(* Logix 5000 project; controller PRU vendor 1 type 14 code 107 rev 20.13; software revision 20.01; part 17 of 17 *)
(* tags used below, declared in another part *)
   AFI : BOOL;
   AlarmMaster : DINT;
   ALL_SHUTDOWN_FAULTS_IOK : BOOL;
   AUTO_FWD_CMD_GON : BOOL;
   CHANGING_TOTE_1 : BOOL;
   DRYER_MODE_AUTO : BOOL;
   ENCODER_ACC : REAL;
   FEED_DWELL_DEG : INT;
   FEED_IS_DWELLING : BOOL;
   FEED_SHOT_ENABLE_Enabled : BOOL;
   FEED_SHOT_ENABLE_GON : BOOL;
   FEED_SHOT_ENABLE_GON_Tmr : TIMER;
   FEED_SHOT_ENABLE_GON_TmrONS1 : BOOL;
   FEED_SHOT_ENABLE_GON_TmrONS2 : BOOL;
   FEED_SHOT_ENABLE_ONS : BOOL;
   FEED_SHOT_ENABLE_ONSN : BOOL;
   FEED_SHOT_ENABLE_SS : BOOL;
   FEED_SHOT_ENABLE_SSN : BOOL;
   FEED_TIME : REAL;
   FEED_TIME_OFF_SEC : REAL;
   FEED_TIME_ON_SEC : REAL;
   FEED_UNWIND_THRESHOLD : INT;
   FIRST_CYCLE : BOOL;
   FWD_SCAN_COUNT : DINT;
   FWD_SCAN_COUNTING : DINT;
   FWD_SCAN_SEC : REAL;
   HMI_MIX_REV_PRESET : DINT;
   KPI : KPI;
   KPI_EnergyResetPB : BOOL;
   MIDNIGHT : BOOL;
   MIX_MODE_TIMEBASE : BOOL;
   PROCESS_SEQUENCER : INT;
   PRU_ShotEnabledTestTmr : TIMER;
   PRU_ShotEnabledTestTmrONS : BOOL;
   PRU_Status_Data : PLCStatusData;
   PYRO_CYCLE_TIME_RESET_ONS : BOOL;
   PYRO_CYCLE_TIME_RESET_SS : BOOL;
   PYRO_FWD_RUN_IOK : BOOL;
   PYRO_FWD_TON : TIMER;
   SET_PYRO_SPEED_TO_ZERO : BOOL;
   STANDBY_MODE_ION : BOOL;
   TOTAL_SCAN_COUNT : DINT;
   TOTAL_SCAN_COUNTING : DINT;
   TOTAL_SCAN_SEC : REAL;
   UTL_Status_Data : PLCStatusData;
   VFD_1_Tot : EnergyTot;   // Left Dryer
   VFD_2_Tot : EnergyTot;   // Right Dryer
   VFD_3_Tot : EnergyTot;   // Cooling Screw
   VFDS_BON : BOOL;   // DRYER VFDs HAVE BEEN COMMANDED ON FOR 1 SECOND.
   Z1L1_Tot : EnergyTot;
   Z1L2_Tot : EnergyTot;
   Z1L3_Tot : EnergyTot;
   Z2L1_Tot : EnergyTot;
   Z2L2_Tot : EnergyTot;
   Z2L3_Tot : EnergyTot;
   Z3L1_Tot : EnergyTot;
   Z3L2_Tot : EnergyTot;
   Z3L3_Tot : EnergyTot;
   Z4L1_Tot : EnergyTot;
   Z5L2_Tot : EnergyTot;
   Z6L3_Tot : EnergyTot;
   Z7L1_Tot : EnergyTot;
   Z8L2_Tot : EnergyTot;
   Z9L3_Tot : EnergyTot;
(* SCREW_CONTROL, continued *)

ROUTINE FEED_CONTROL   (* ladder *)
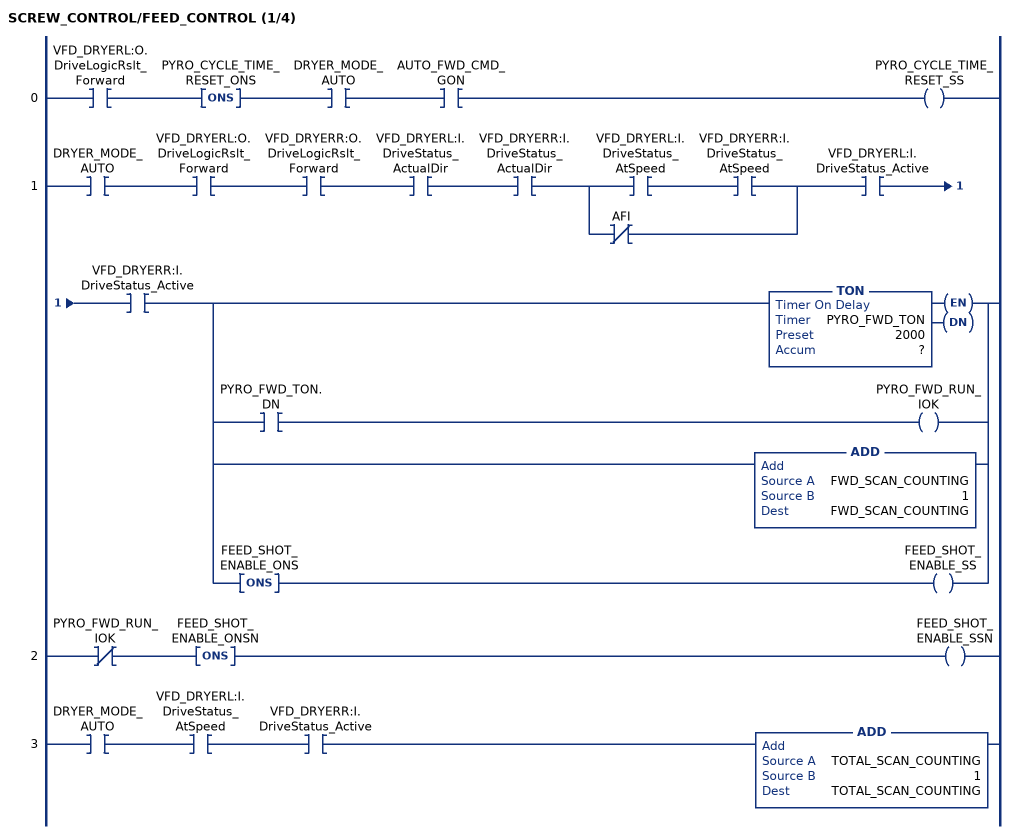
   0: XIC(VFD_DRYERL:O.DriveLogicRslt_Forward)ONS(PYRO_CYCLE_TIME_RESET_ONS)XIC(DRYER_MODE_AUTO)XIC(AUTO_FWD_CMD_GON)OTE(PYRO_CYCLE_TIME_RESET_SS);
   1: XIC(DRYER_MODE_AUTO)XIC(VFD_DRYERL:O.DriveLogicRslt_Forward)XIC(VFD_DRYERR:O.DriveLogicRslt_Forward)XIC(VFD_DRYERL:I.DriveStatus_ActualDir)XIC(VFD_DRYERR:I.DriveStatus_ActualDir)[XIC(VFD_DRYERL:I.DriveStatus_AtSpeed) XIC(VFD_DRYERR:I.DriveStatus_AtSpeed) ,XIO(AFI) ]XIC(VFD_DRYERL:I.DriveStatus_Active)XIC(VFD_DRYERR:I.DriveStatus_Active)[TON(PYRO_FWD_TON,?,?) ,XIC(PYRO_FWD_TON.DN) OTE(PYRO_FWD_RUN_IOK) ,ADD(FWD_SCAN_COUNTING,1,FWD_SCAN_COUNTING) ,ONS(FEED_SHOT_ENABLE_ONS) OTE(FEED_SHOT_ENABLE_SS) ];
   2: XIO(PYRO_FWD_RUN_IOK)ONS(FEED_SHOT_ENABLE_ONSN)OTE(FEED_SHOT_ENABLE_SSN);
   3: XIC(DRYER_MODE_AUTO)XIC(VFD_DRYERL:I.DriveStatus_AtSpeed)XIC(VFD_DRYERR:I.DriveStatus_Active)ADD(TOTAL_SCAN_COUNTING,1,TOTAL_SCAN_COUNTING);
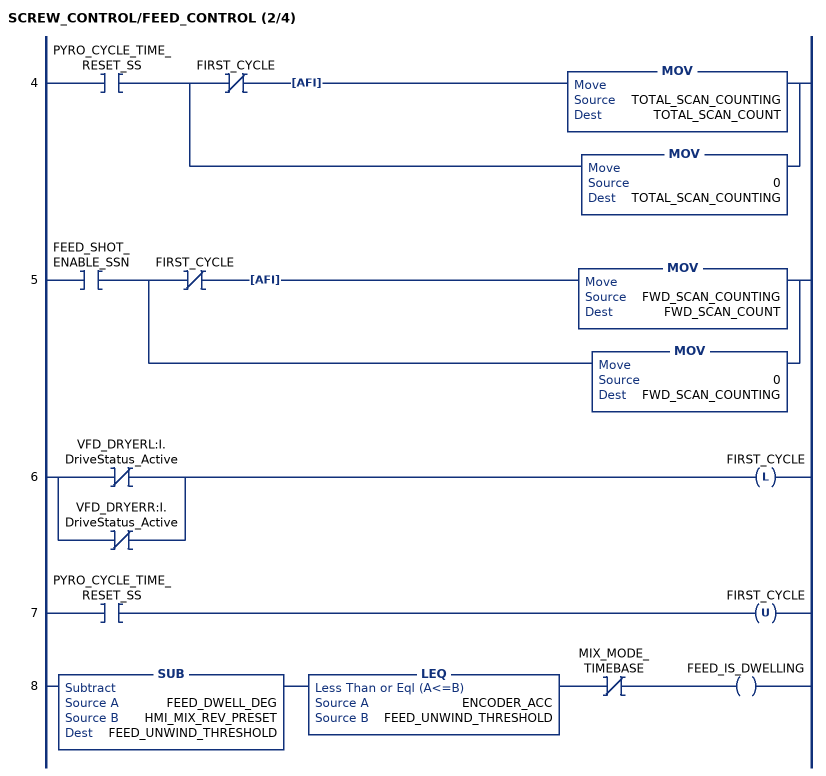
   4: XIC(PYRO_CYCLE_TIME_RESET_SS)[XIO(FIRST_CYCLE) AFI() MOV(TOTAL_SCAN_COUNTING,TOTAL_SCAN_COUNT) ,MOV(0,TOTAL_SCAN_COUNTING) ];
   5: XIC(FEED_SHOT_ENABLE_SSN)[XIO(FIRST_CYCLE) AFI() MOV(FWD_SCAN_COUNTING,FWD_SCAN_COUNT) ,MOV(0,FWD_SCAN_COUNTING) ];
   6: [XIO(VFD_DRYERL:I.DriveStatus_Active) ,XIO(VFD_DRYERR:I.DriveStatus_Active) ]OTL(FIRST_CYCLE);
   7: XIC(PYRO_CYCLE_TIME_RESET_SS)OTU(FIRST_CYCLE);
   8: SUB(FEED_DWELL_DEG,HMI_MIX_REV_PRESET,FEED_UNWIND_THRESHOLD)LEQ(ENCODER_ACC,FEED_UNWIND_THRESHOLD)XIO(MIX_MODE_TIMEBASE)OTE(FEED_IS_DWELLING);
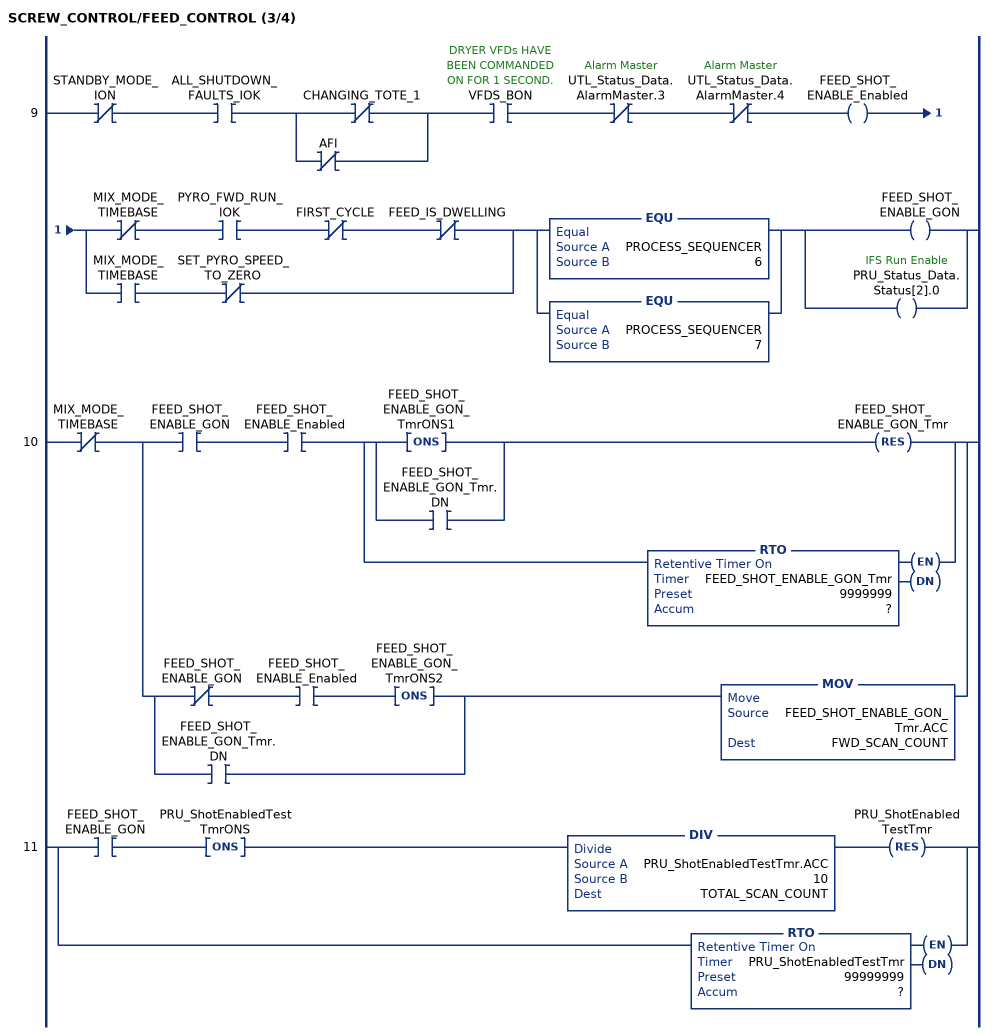
   9: XIO(STANDBY_MODE_ION)XIC(ALL_SHUTDOWN_FAULTS_IOK)[XIO(CHANGING_TOTE_1) ,XIO(AFI) ]XIC(VFDS_BON)XIO(UTL_Status_Data.AlarmMaster.3)XIO(UTL_Status_Data.AlarmMaster.4)OTE(FEED_SHOT_ENABLE_Enabled)[XIO(MIX_MODE_TIMEBASE) XIC(PYRO_FWD_RUN_IOK) XIO(FIRST_CYCLE) XIO(FEED_IS_DWELLING) ,XIC(MIX_MODE_TIMEBASE) XIO(SET_PYRO_SPEED_TO_ZERO) ][EQU(PROCESS_SEQUENCER,6) ,EQU(PROCESS_SEQUENCER,7) ][OTE(FEED_SHOT_ENABLE_GON) ,OTE(PRU_Status_Data.Status[2].0) ];
   10: XIO(MIX_MODE_TIMEBASE)[XIC(FEED_SHOT_ENABLE_GON) XIC(FEED_SHOT_ENABLE_Enabled) [[ONS(FEED_SHOT_ENABLE_GON_TmrONS1) ,XIC(FEED_SHOT_ENABLE_GON_Tmr.DN) ] RES(FEED_SHOT_ENABLE_GON_Tmr) ,RTO(FEED_SHOT_ENABLE_GON_Tmr,?,?) ] ,[XIO(FEED_SHOT_ENABLE_GON) XIC(FEED_SHOT_ENABLE_Enabled) ONS(FEED_SHOT_ENABLE_GON_TmrONS2) ,XIC(FEED_SHOT_ENABLE_GON_Tmr.DN) ] MOV(FEED_SHOT_ENABLE_GON_Tmr.ACC,FWD_SCAN_COUNT) ];
   11: [XIC(FEED_SHOT_ENABLE_GON) ONS(PRU_ShotEnabledTestTmrONS) DIV(PRU_ShotEnabledTestTmr.ACC,10,TOTAL_SCAN_COUNT) RES(PRU_ShotEnabledTestTmr) ,RTO(PRU_ShotEnabledTestTmr,?,?) ];
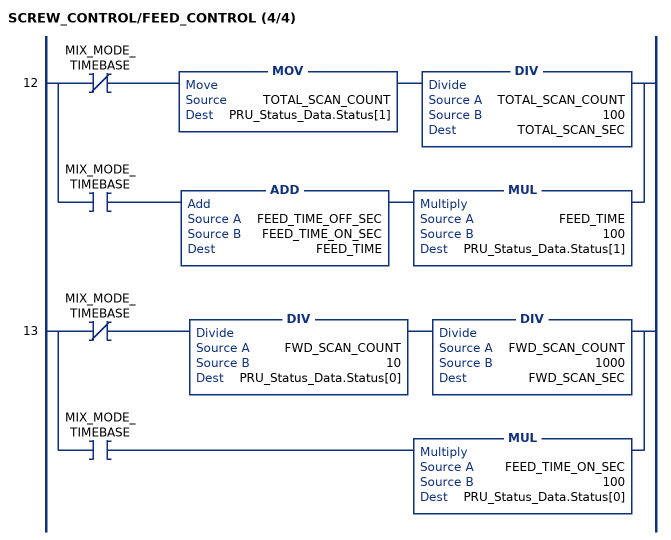
   12: [XIO(MIX_MODE_TIMEBASE) MOV(TOTAL_SCAN_COUNT,PRU_Status_Data.Status[1]) DIV(TOTAL_SCAN_COUNT,100,TOTAL_SCAN_SEC) ,XIC(MIX_MODE_TIMEBASE) ADD(FEED_TIME_OFF_SEC,FEED_TIME_ON_SEC,FEED_TIME) MUL(FEED_TIME,100,PRU_Status_Data.Status[1]) ];
   13: [XIO(MIX_MODE_TIMEBASE) DIV(FWD_SCAN_COUNT,10,PRU_Status_Data.Status[0]) DIV(FWD_SCAN_COUNT,1000,FWD_SCAN_SEC) ,XIC(MIX_MODE_TIMEBASE) MUL(FEED_TIME_ON_SEC,100,PRU_Status_Data.Status[0]) ];
END_ROUTINE
END_PROGRAM

PROGRAM Totalizers   (* main routine MainRoutine *)
VAR
   AITot_VFD1 : AI_Totalizer := (Input := 5.23152, SampleTimerSP := 1, TimeBase := 3, MinimumInc := 1.0, IDP := 2, RollOver := 999999999, NonResetTotal := 618304, TodayTotal := 1933, YestTotal := 4297, ResetTotal := 497307);
   AITot_VFD2 : AI_Totalizer := (Input := 5.3976, SampleTimerSP := 1, TimeBase := 3, MinimumInc := 1.0, IDP := 2, RollOver := 999999999, NonResetTotal := 632266, TodayTotal := 1996, YestTotal := 4422, ResetTotal := 509519);
   AITot_VFD3 : AI_Totalizer := (Input := 1.5943679, SampleTimerSP := 1, TimeBase := 3, MinimumInc := 1.0, IDP := 2, RollOver := 999999999, NonResetTotal := 173015, TodayTotal := 587, YestTotal := 1277, ResetTotal := 140164);
   AITot_Z1L1 : AI_Totalizer := (Input := 1.689711, SampleTimerSP := 1, TimeBase := 3, MinimumInc := 1.0, IDP := 2, RollOver := 999999999, NonResetTotal := 472353, TodayTotal := 130, YestTotal := 3764, ResetTotal := 404849);
   AITot_Z1L2 : AI_Totalizer := (Input := 0.03052023, SampleTimerSP := 1, TimeBase := 3, MinimumInc := 1.0, IDP := 2, RollOver := 999999999, NonResetTotal := 457837, TodayTotal := 130, YestTotal := 3741, ResetTotal := 457837);
   AITot_Z1L3 : AI_Totalizer := (Input := 0.03052023, SampleTimerSP := 1, TimeBase := 3, MinimumInc := 1.0, IDP := 2, RollOver := 999999999, NonResetTotal := 456822, TodayTotal := 160, YestTotal := 4321, ResetTotal := 390415);
   AITot_Z2L1 : AI_Totalizer := (Input := 1.2069364, SampleTimerSP := 1, TimeBase := 3, MinimumInc := 1.0, IDP := 2, RollOver := 999999999, NonResetTotal := 262631, TodayTotal := 198, YestTotal := 2727, ResetTotal := 202203);
   AITot_Z2L2 : AI_Totalizer := (Input := 0.033294797, SampleTimerSP := 1, TimeBase := 3, MinimumInc := 1.0, IDP := 2, RollOver := 999999999, NonResetTotal := 260774, TodayTotal := 195, YestTotal := 2658, ResetTotal := 201494);
   AITot_Z2L3 : AI_Totalizer := (Input := 1.2873988, SampleTimerSP := 1, TimeBase := 3, MinimumInc := 1.0, IDP := 2, RollOver := 999999999, NonResetTotal := 261254, TodayTotal := 195, YestTotal := 2685, ResetTotal := 201639);
   AITot_Z3L1 : AI_Totalizer := (Input := 0.8323699, SampleTimerSP := 1, TimeBase := 3, MinimumInc := 1.0, IDP := 2, RollOver := 999999999, NonResetTotal := 191746, TodayTotal := 428, YestTotal := 2124, ResetTotal := 154486);
   AITot_Z3L2 : AI_Totalizer := (Input := 0.88508666, SampleTimerSP := 1, TimeBase := 3, MinimumInc := 1.0, IDP := 2, RollOver := 999999999, NonResetTotal := 197557, TodayTotal := 352, YestTotal := 1665, ResetTotal := 160053);
   AITot_Z3L3 : AI_Totalizer := (Input := 0.59930634, SampleTimerSP := 1, TimeBase := 3, MinimumInc := 1.0, IDP := 2, RollOver := 999999999, NonResetTotal := 197140, TodayTotal := 341, YestTotal := 1652, ResetTotal := 160368);
   AITot_Z4L1 : AI_Totalizer := (Input := 0.88508666, SampleTimerSP := 1, TimeBase := 3, MinimumInc := 1.0, IDP := 2, RollOver := 999999999, NonResetTotal := 314322, TodayTotal := 64, YestTotal := 1698, ResetTotal := 297528);
   AITot_Z5L2 : AI_Totalizer := (Input := 0.03052023, SampleTimerSP := 1, TimeBase := 3, MinimumInc := 1.0, IDP := 2, RollOver := 999999999, NonResetTotal := 574405, TodayTotal := 368, YestTotal := 5145, ResetTotal := 490444);
   AITot_Z6L3 : AI_Totalizer := (Input := 0.30797687, SampleTimerSP := 1, TimeBase := 3, MinimumInc := 1.0, IDP := 2, RollOver := 999999999, NonResetTotal := 104261, TodayTotal := 197, YestTotal := 2603, ResetTotal := 99809);
   AITot_Z7L1 : AI_Totalizer := (Input := 0.03052023, SampleTimerSP := 1, TimeBase := 3, MinimumInc := 1.0, IDP := 2, RollOver := 999999999, NonResetTotal := 390081, TodayTotal := 454, YestTotal := 4326, ResetTotal := 301917);
   AITot_Z8L2 : AI_Totalizer := (Input := 5.041387, SampleTimerSP := 1, TimeBase := 3, MinimumInc := 1.0, IDP := 2, RollOver := 999999999, NonResetTotal := 336435, TodayTotal := 1724, YestTotal := 5854, ResetTotal := 321398);
   AITot_Z9L3 : AI_Totalizer := (Input := 5.6684394, SampleTimerSP := 1, TimeBase := 3, MinimumInc := 1.0, IDP := 2, RollOver := 999999999, NonResetTotal := 446178, TodayTotal := 1624, YestTotal := 4125, ResetTotal := 368110);
   ResetTotalizersONS : BOOL;
END_VAR

ROUTINE MainRoutine   (* ladder *)
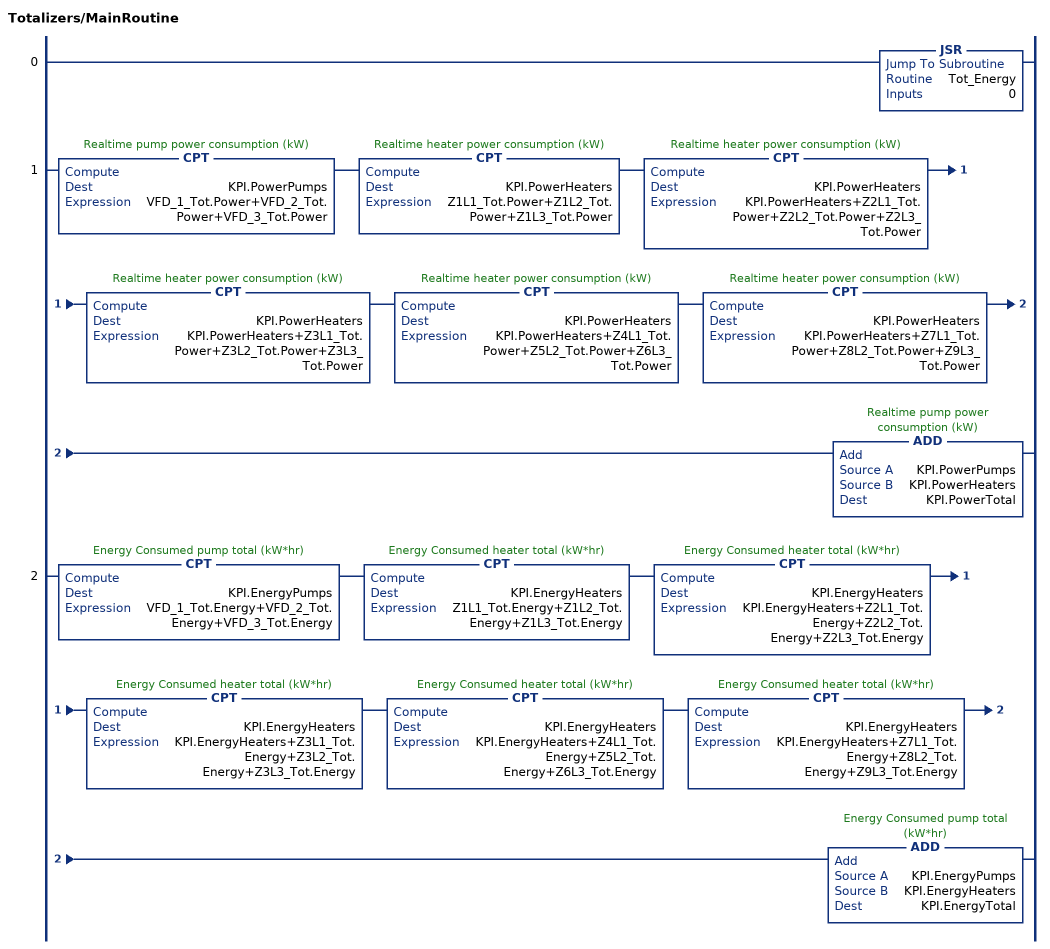
   0: JSR(Tot_Energy,0);
   1: CPT(KPI.PowerPumps,VFD_1_Tot.Power+VFD_2_Tot.Power+VFD_3_Tot.Power)CPT(KPI.PowerHeaters,Z1L1_Tot.Power+Z1L2_Tot.Power+Z1L3_Tot.Power)CPT(KPI.PowerHeaters,KPI.PowerHeaters+Z2L1_Tot.Power+Z2L2_Tot.Power+Z2L3_Tot.Power)CPT(KPI.PowerHeaters,KPI.PowerHeaters+Z3L1_Tot.Power+Z3L2_Tot.Power+Z3L3_Tot.Power)CPT(KPI.PowerHeaters,KPI.PowerHeaters+Z4L1_Tot.Power+Z5L2_Tot.Power+Z6L3_Tot.Power)CPT(KPI.PowerHeaters,KPI.PowerHeaters+Z7L1_Tot.Power+Z8L2_Tot.Power+Z9L3_Tot.Power)ADD(KPI.PowerPumps,KPI.PowerHeaters,KPI.PowerTotal);
   2: CPT(KPI.EnergyPumps,VFD_1_Tot.Energy+VFD_2_Tot.Energy+VFD_3_Tot.Energy)CPT(KPI.EnergyHeaters,Z1L1_Tot.Energy+Z1L2_Tot.Energy+Z1L3_Tot.Energy)CPT(KPI.EnergyHeaters,KPI.EnergyHeaters+Z2L1_Tot.Energy+Z2L2_Tot.Energy+Z2L3_Tot.Energy)CPT(KPI.EnergyHeaters,KPI.EnergyHeaters+Z3L1_Tot.Energy+Z3L2_Tot.Energy+Z3L3_Tot.Energy)CPT(KPI.EnergyHeaters,KPI.EnergyHeaters+Z4L1_Tot.Energy+Z5L2_Tot.Energy+Z6L3_Tot.Energy)CPT(KPI.EnergyHeaters,KPI.EnergyHeaters+Z7L1_Tot.Energy+Z8L2_Tot.Energy+Z9L3_Tot.Energy)ADD(KPI.EnergyPumps,KPI.EnergyHeaters,KPI.EnergyTotal);
END_ROUTINE

ROUTINE Tot_Energy   (* ladder *)
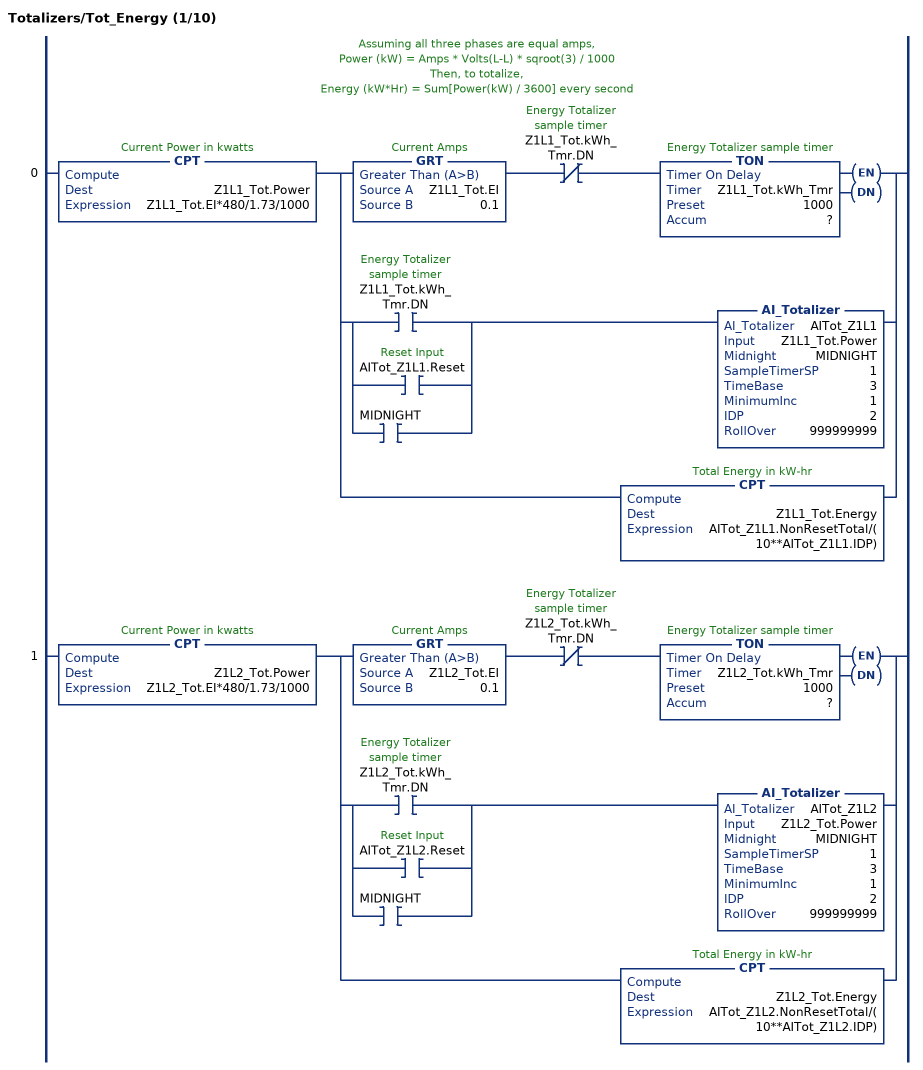
   // Assuming all three phases are equal amps,
   // Power (kW) = Amps * Volts(L-L) * sqroot(3) / 1000
   // Then, to totalize,
   // Energy (kW*Hr) = Sum[Power(kW) / 3600] every second
   0: CPT(Z1L1_Tot.Power,Z1L1_Tot.EI*480/1.73/1000)[GRT(Z1L1_Tot.EI,0.1) XIO(Z1L1_Tot.kWh_Tmr.DN) TON(Z1L1_Tot.kWh_Tmr,?,?) ,[XIC(Z1L1_Tot.kWh_Tmr.DN) ,XIC(AITot_Z1L1.Reset) ,XIC(MIDNIGHT) ] AI_Totalizer(AITot_Z1L1,Z1L1_Tot.Power,MIDNIGHT,1,3,1,2,999999999) ,CPT(Z1L1_Tot.Energy,AITot_Z1L1.NonResetTotal/(10**AITot_Z1L1.IDP)) ];
   1: CPT(Z1L2_Tot.Power,Z1L2_Tot.EI*480/1.73/1000)[GRT(Z1L2_Tot.EI,0.1) XIO(Z1L2_Tot.kWh_Tmr.DN) TON(Z1L2_Tot.kWh_Tmr,?,?) ,[XIC(Z1L2_Tot.kWh_Tmr.DN) ,XIC(AITot_Z1L2.Reset) ,XIC(MIDNIGHT) ] AI_Totalizer(AITot_Z1L2,Z1L2_Tot.Power,MIDNIGHT,1,3,1,2,999999999) ,CPT(Z1L2_Tot.Energy,AITot_Z1L2.NonResetTotal/(10**AITot_Z1L2.IDP)) ];
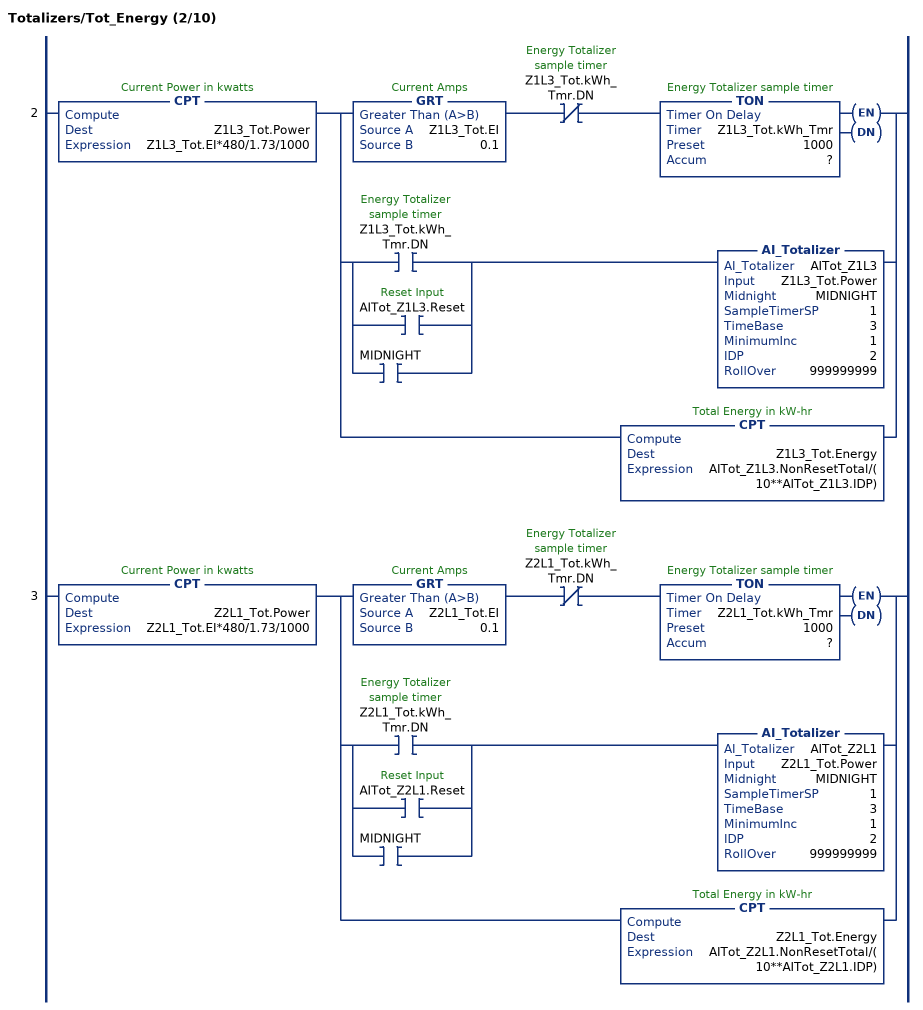
   2: CPT(Z1L3_Tot.Power,Z1L3_Tot.EI*480/1.73/1000)[GRT(Z1L3_Tot.EI,0.1) XIO(Z1L3_Tot.kWh_Tmr.DN) TON(Z1L3_Tot.kWh_Tmr,?,?) ,[XIC(Z1L3_Tot.kWh_Tmr.DN) ,XIC(AITot_Z1L3.Reset) ,XIC(MIDNIGHT) ] AI_Totalizer(AITot_Z1L3,Z1L3_Tot.Power,MIDNIGHT,1,3,1,2,999999999) ,CPT(Z1L3_Tot.Energy,AITot_Z1L3.NonResetTotal/(10**AITot_Z1L3.IDP)) ];
   3: CPT(Z2L1_Tot.Power,Z2L1_Tot.EI*480/1.73/1000)[GRT(Z2L1_Tot.EI,0.1) XIO(Z2L1_Tot.kWh_Tmr.DN) TON(Z2L1_Tot.kWh_Tmr,?,?) ,[XIC(Z2L1_Tot.kWh_Tmr.DN) ,XIC(AITot_Z2L1.Reset) ,XIC(MIDNIGHT) ] AI_Totalizer(AITot_Z2L1,Z2L1_Tot.Power,MIDNIGHT,1,3,1,2,999999999) ,CPT(Z2L1_Tot.Energy,AITot_Z2L1.NonResetTotal/(10**AITot_Z2L1.IDP)) ];
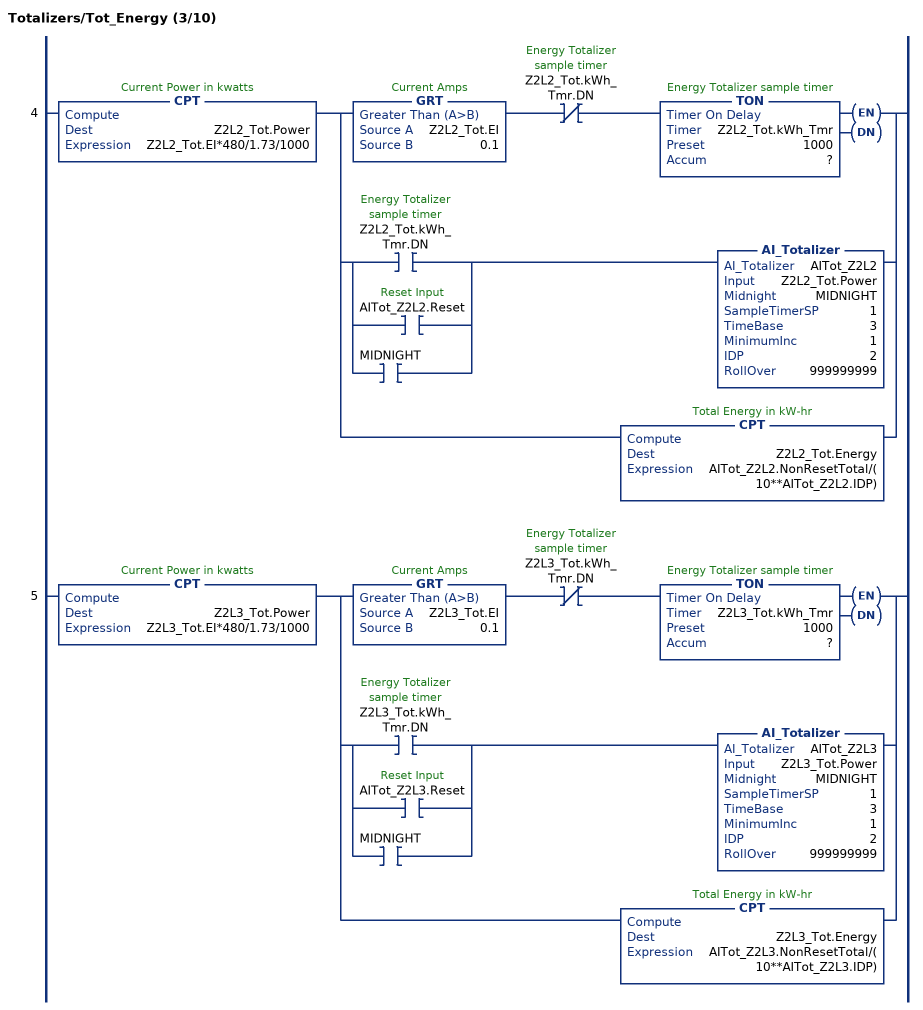
   4: CPT(Z2L2_Tot.Power,Z2L2_Tot.EI*480/1.73/1000)[GRT(Z2L2_Tot.EI,0.1) XIO(Z2L2_Tot.kWh_Tmr.DN) TON(Z2L2_Tot.kWh_Tmr,?,?) ,[XIC(Z2L2_Tot.kWh_Tmr.DN) ,XIC(AITot_Z2L2.Reset) ,XIC(MIDNIGHT) ] AI_Totalizer(AITot_Z2L2,Z2L2_Tot.Power,MIDNIGHT,1,3,1,2,999999999) ,CPT(Z2L2_Tot.Energy,AITot_Z2L2.NonResetTotal/(10**AITot_Z2L2.IDP)) ];
   5: CPT(Z2L3_Tot.Power,Z2L3_Tot.EI*480/1.73/1000)[GRT(Z2L3_Tot.EI,0.1) XIO(Z2L3_Tot.kWh_Tmr.DN) TON(Z2L3_Tot.kWh_Tmr,?,?) ,[XIC(Z2L3_Tot.kWh_Tmr.DN) ,XIC(AITot_Z2L3.Reset) ,XIC(MIDNIGHT) ] AI_Totalizer(AITot_Z2L3,Z2L3_Tot.Power,MIDNIGHT,1,3,1,2,999999999) ,CPT(Z2L3_Tot.Energy,AITot_Z2L3.NonResetTotal/(10**AITot_Z2L3.IDP)) ];
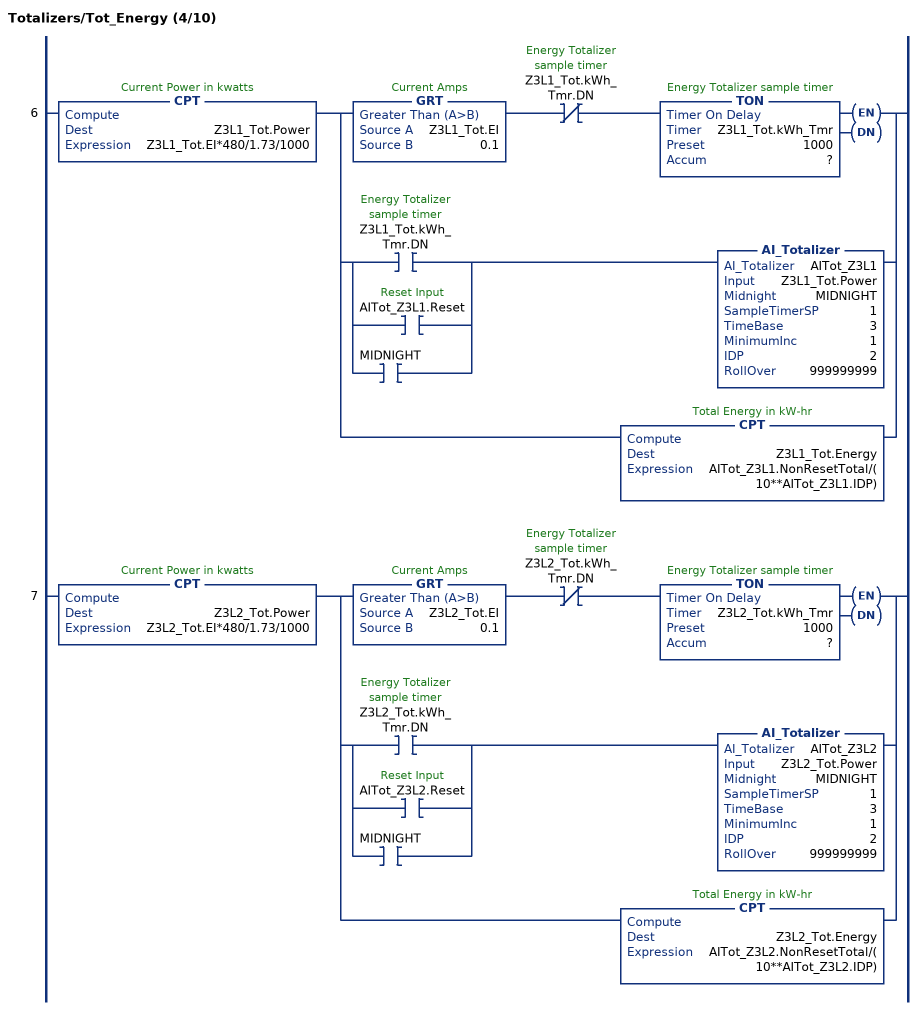
   6: CPT(Z3L1_Tot.Power,Z3L1_Tot.EI*480/1.73/1000)[GRT(Z3L1_Tot.EI,0.1) XIO(Z3L1_Tot.kWh_Tmr.DN) TON(Z3L1_Tot.kWh_Tmr,?,?) ,[XIC(Z3L1_Tot.kWh_Tmr.DN) ,XIC(AITot_Z3L1.Reset) ,XIC(MIDNIGHT) ] AI_Totalizer(AITot_Z3L1,Z3L1_Tot.Power,MIDNIGHT,1,3,1,2,999999999) ,CPT(Z3L1_Tot.Energy,AITot_Z3L1.NonResetTotal/(10**AITot_Z3L1.IDP)) ];
   7: CPT(Z3L2_Tot.Power,Z3L2_Tot.EI*480/1.73/1000)[GRT(Z3L2_Tot.EI,0.1) XIO(Z3L2_Tot.kWh_Tmr.DN) TON(Z3L2_Tot.kWh_Tmr,?,?) ,[XIC(Z3L2_Tot.kWh_Tmr.DN) ,XIC(AITot_Z3L2.Reset) ,XIC(MIDNIGHT) ] AI_Totalizer(AITot_Z3L2,Z3L2_Tot.Power,MIDNIGHT,1,3,1,2,999999999) ,CPT(Z3L2_Tot.Energy,AITot_Z3L2.NonResetTotal/(10**AITot_Z3L2.IDP)) ];
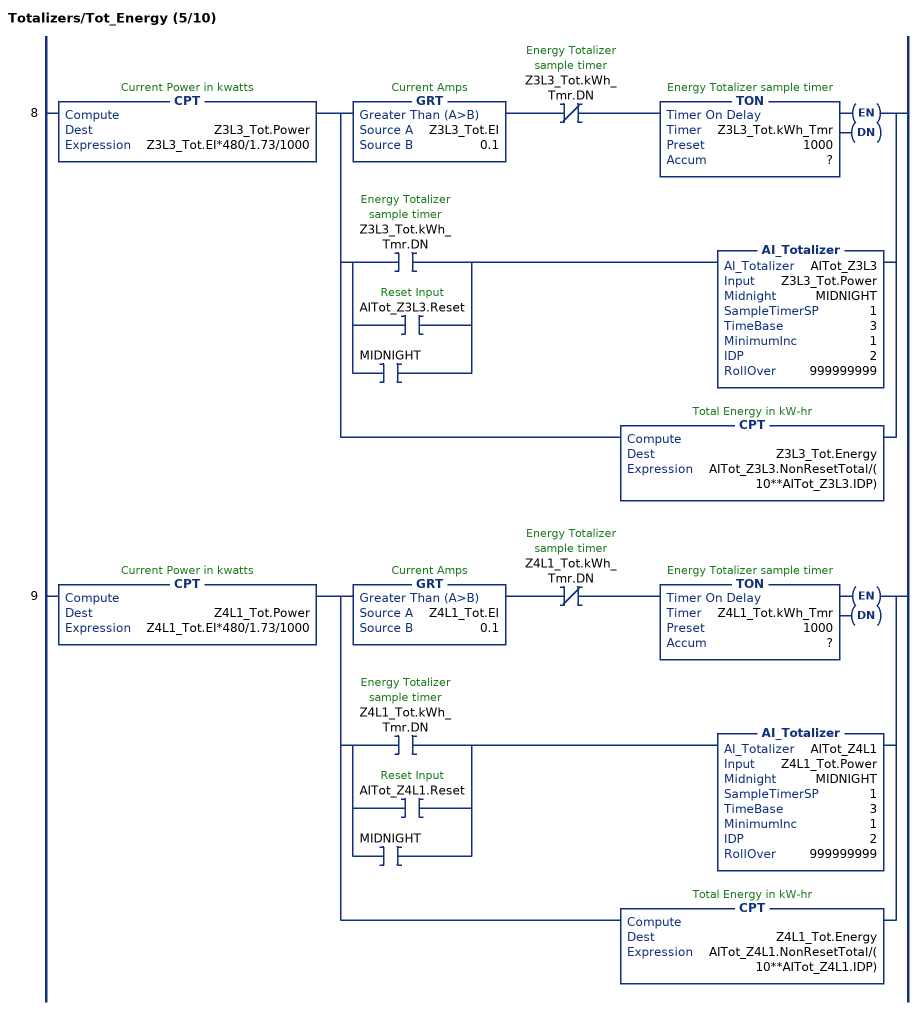
   8: CPT(Z3L3_Tot.Power,Z3L3_Tot.EI*480/1.73/1000)[GRT(Z3L3_Tot.EI,0.1) XIO(Z3L3_Tot.kWh_Tmr.DN) TON(Z3L3_Tot.kWh_Tmr,?,?) ,[XIC(Z3L3_Tot.kWh_Tmr.DN) ,XIC(AITot_Z3L3.Reset) ,XIC(MIDNIGHT) ] AI_Totalizer(AITot_Z3L3,Z3L3_Tot.Power,MIDNIGHT,1,3,1,2,999999999) ,CPT(Z3L3_Tot.Energy,AITot_Z3L3.NonResetTotal/(10**AITot_Z3L3.IDP)) ];
   9: CPT(Z4L1_Tot.Power,Z4L1_Tot.EI*480/1.73/1000)[GRT(Z4L1_Tot.EI,0.1) XIO(Z4L1_Tot.kWh_Tmr.DN) TON(Z4L1_Tot.kWh_Tmr,?,?) ,[XIC(Z4L1_Tot.kWh_Tmr.DN) ,XIC(AITot_Z4L1.Reset) ,XIC(MIDNIGHT) ] AI_Totalizer(AITot_Z4L1,Z4L1_Tot.Power,MIDNIGHT,1,3,1,2,999999999) ,CPT(Z4L1_Tot.Energy,AITot_Z4L1.NonResetTotal/(10**AITot_Z4L1.IDP)) ];
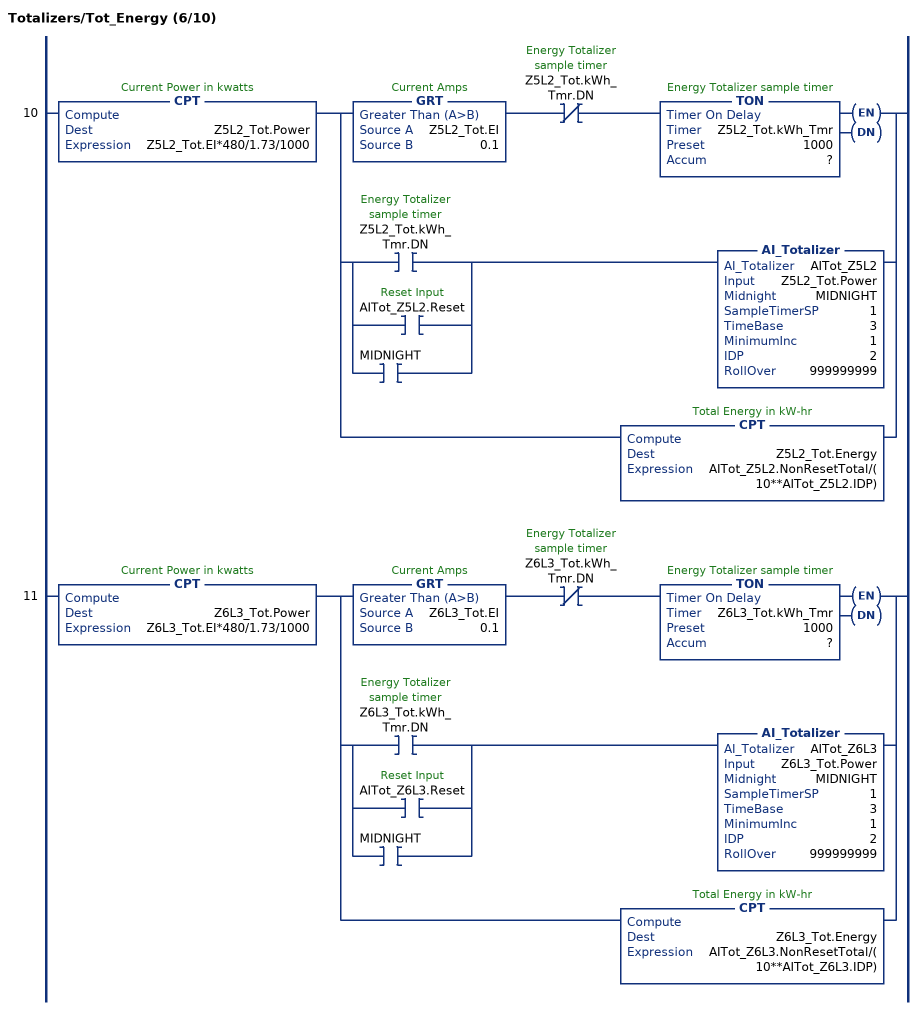
   10: CPT(Z5L2_Tot.Power,Z5L2_Tot.EI*480/1.73/1000)[GRT(Z5L2_Tot.EI,0.1) XIO(Z5L2_Tot.kWh_Tmr.DN) TON(Z5L2_Tot.kWh_Tmr,?,?) ,[XIC(Z5L2_Tot.kWh_Tmr.DN) ,XIC(AITot_Z5L2.Reset) ,XIC(MIDNIGHT) ] AI_Totalizer(AITot_Z5L2,Z5L2_Tot.Power,MIDNIGHT,1,3,1,2,999999999) ,CPT(Z5L2_Tot.Energy,AITot_Z5L2.NonResetTotal/(10**AITot_Z5L2.IDP)) ];
   11: CPT(Z6L3_Tot.Power,Z6L3_Tot.EI*480/1.73/1000)[GRT(Z6L3_Tot.EI,0.1) XIO(Z6L3_Tot.kWh_Tmr.DN) TON(Z6L3_Tot.kWh_Tmr,?,?) ,[XIC(Z6L3_Tot.kWh_Tmr.DN) ,XIC(AITot_Z6L3.Reset) ,XIC(MIDNIGHT) ] AI_Totalizer(AITot_Z6L3,Z6L3_Tot.Power,MIDNIGHT,1,3,1,2,999999999) ,CPT(Z6L3_Tot.Energy,AITot_Z6L3.NonResetTotal/(10**AITot_Z6L3.IDP)) ];
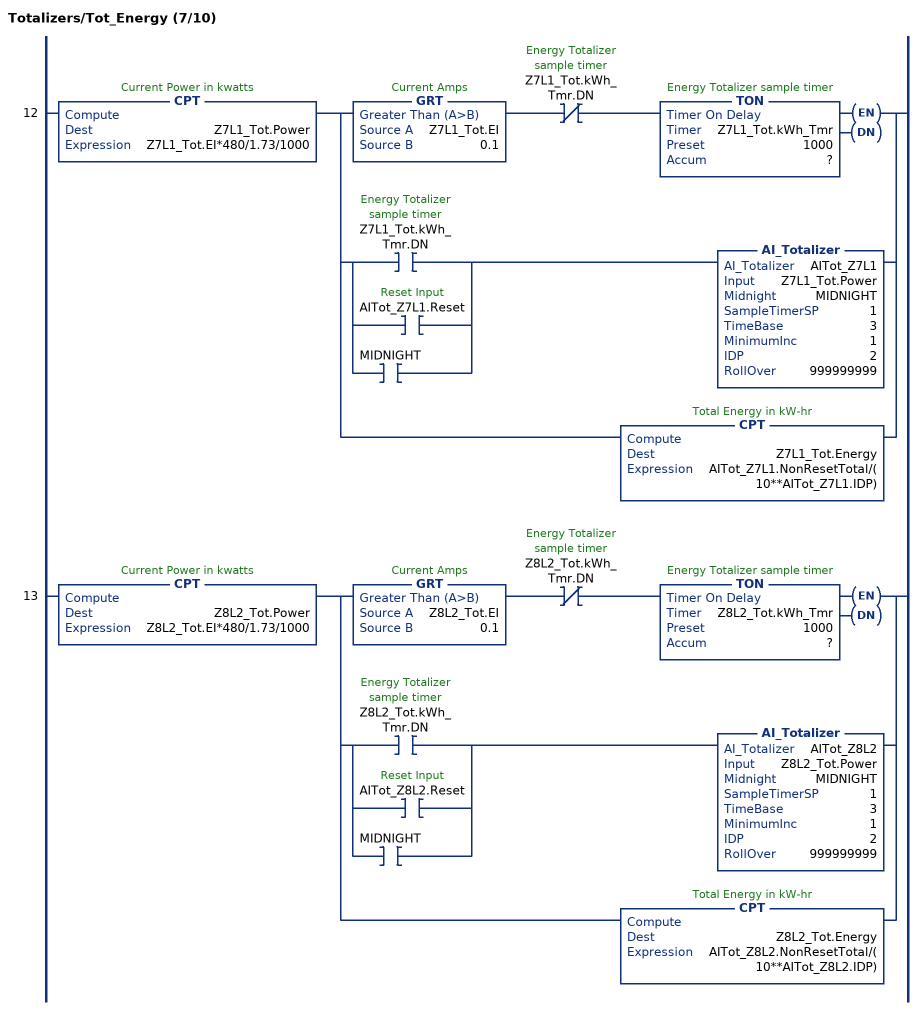
   12: CPT(Z7L1_Tot.Power,Z7L1_Tot.EI*480/1.73/1000)[GRT(Z7L1_Tot.EI,0.1) XIO(Z7L1_Tot.kWh_Tmr.DN) TON(Z7L1_Tot.kWh_Tmr,?,?) ,[XIC(Z7L1_Tot.kWh_Tmr.DN) ,XIC(AITot_Z7L1.Reset) ,XIC(MIDNIGHT) ] AI_Totalizer(AITot_Z7L1,Z7L1_Tot.Power,MIDNIGHT,1,3,1,2,999999999) ,CPT(Z7L1_Tot.Energy,AITot_Z7L1.NonResetTotal/(10**AITot_Z7L1.IDP)) ];
   13: CPT(Z8L2_Tot.Power,Z8L2_Tot.EI*480/1.73/1000)[GRT(Z8L2_Tot.EI,0.1) XIO(Z8L2_Tot.kWh_Tmr.DN) TON(Z8L2_Tot.kWh_Tmr,?,?) ,[XIC(Z8L2_Tot.kWh_Tmr.DN) ,XIC(AITot_Z8L2.Reset) ,XIC(MIDNIGHT) ] AI_Totalizer(AITot_Z8L2,Z8L2_Tot.Power,MIDNIGHT,1,3,1,2,999999999) ,CPT(Z8L2_Tot.Energy,AITot_Z8L2.NonResetTotal/(10**AITot_Z8L2.IDP)) ];
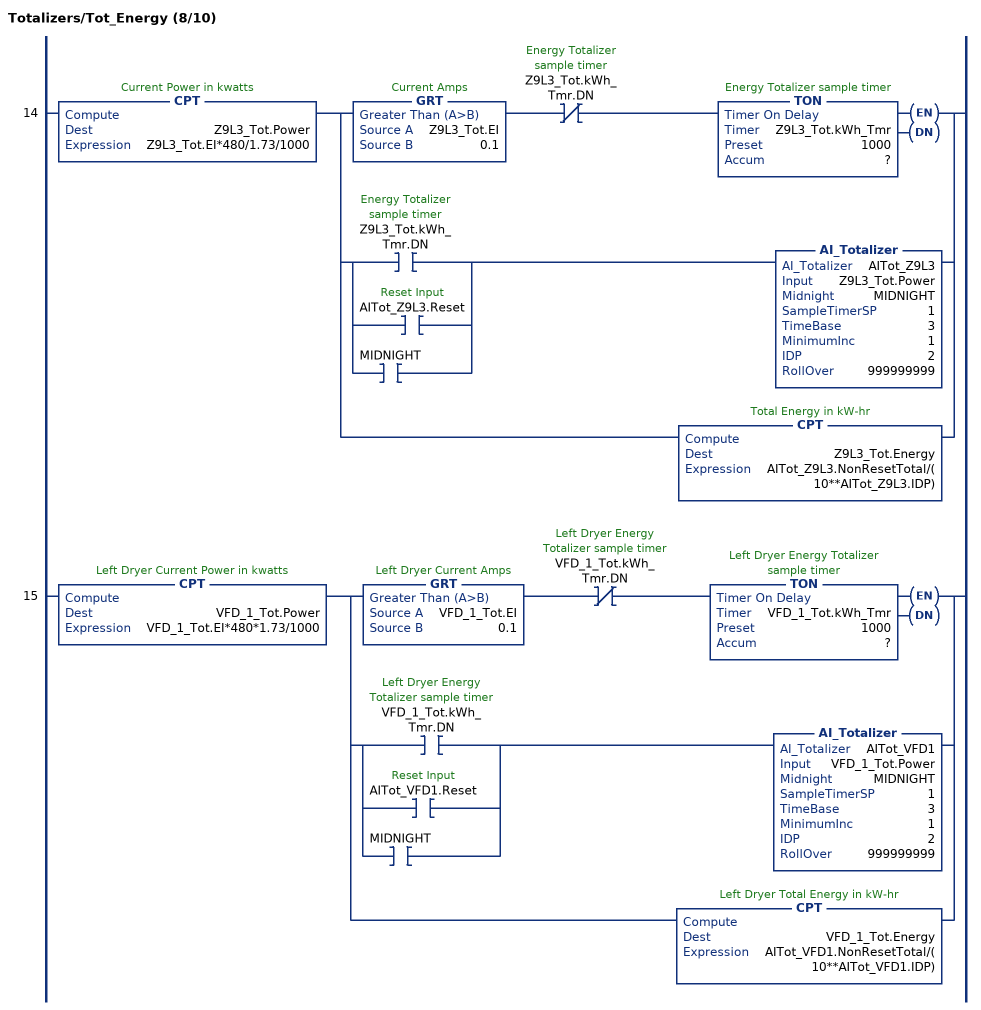
   14: CPT(Z9L3_Tot.Power,Z9L3_Tot.EI*480/1.73/1000)[GRT(Z9L3_Tot.EI,0.1) XIO(Z9L3_Tot.kWh_Tmr.DN) TON(Z9L3_Tot.kWh_Tmr,?,?) ,[XIC(Z9L3_Tot.kWh_Tmr.DN) ,XIC(AITot_Z9L3.Reset) ,XIC(MIDNIGHT) ] AI_Totalizer(AITot_Z9L3,Z9L3_Tot.Power,MIDNIGHT,1,3,1,2,999999999) ,CPT(Z9L3_Tot.Energy,AITot_Z9L3.NonResetTotal/(10**AITot_Z9L3.IDP)) ];
   15: CPT(VFD_1_Tot.Power,VFD_1_Tot.EI*480*1.73/1000)[GRT(VFD_1_Tot.EI,0.1) XIO(VFD_1_Tot.kWh_Tmr.DN) TON(VFD_1_Tot.kWh_Tmr,?,?) ,[XIC(VFD_1_Tot.kWh_Tmr.DN) ,XIC(AITot_VFD1.Reset) ,XIC(MIDNIGHT) ] AI_Totalizer(AITot_VFD1,VFD_1_Tot.Power,MIDNIGHT,1,3,1,2,999999999) ,CPT(VFD_1_Tot.Energy,AITot_VFD1.NonResetTotal/(10**AITot_VFD1.IDP)) ];
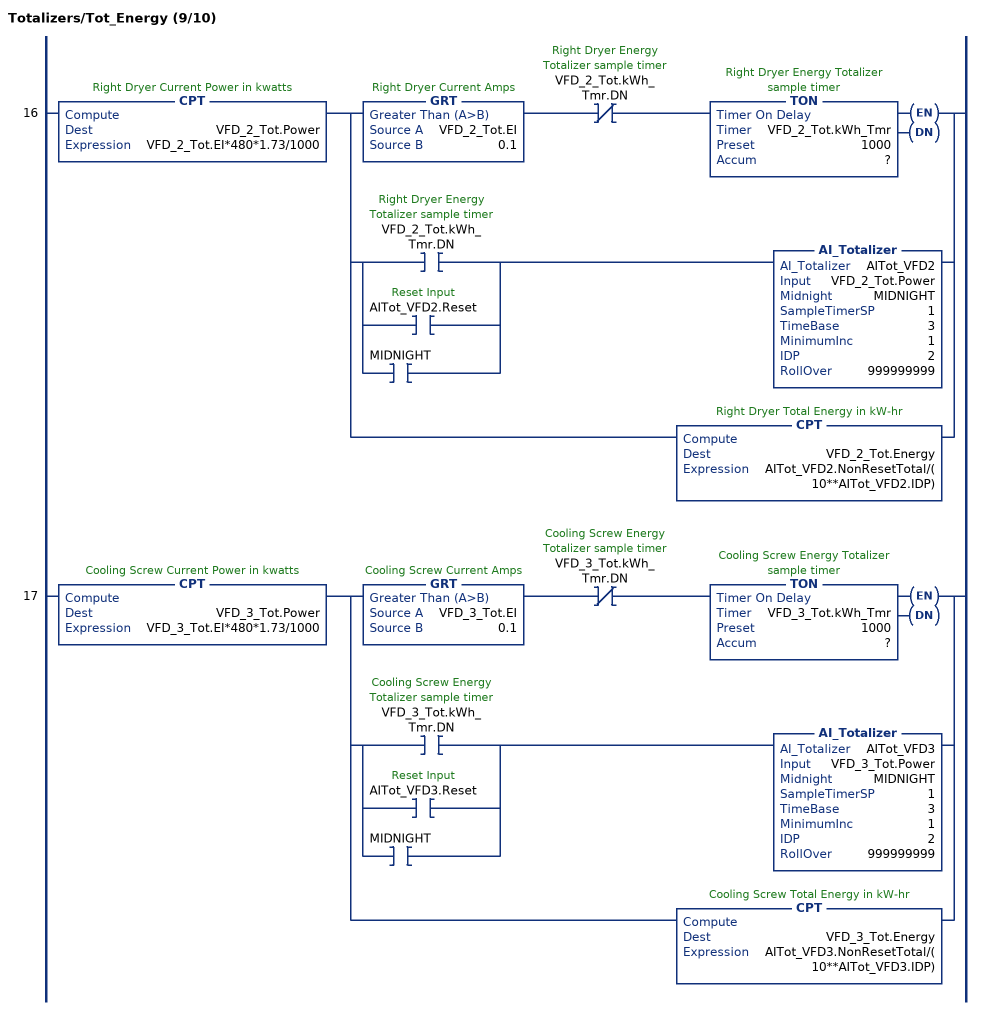
   16: CPT(VFD_2_Tot.Power,VFD_2_Tot.EI*480*1.73/1000)[GRT(VFD_2_Tot.EI,0.1) XIO(VFD_2_Tot.kWh_Tmr.DN) TON(VFD_2_Tot.kWh_Tmr,?,?) ,[XIC(VFD_2_Tot.kWh_Tmr.DN) ,XIC(AITot_VFD2.Reset) ,XIC(MIDNIGHT) ] AI_Totalizer(AITot_VFD2,VFD_2_Tot.Power,MIDNIGHT,1,3,1,2,999999999) ,CPT(VFD_2_Tot.Energy,AITot_VFD2.NonResetTotal/(10**AITot_VFD2.IDP)) ];
   17: CPT(VFD_3_Tot.Power,VFD_3_Tot.EI*480*1.73/1000)[GRT(VFD_3_Tot.EI,0.1) XIO(VFD_3_Tot.kWh_Tmr.DN) TON(VFD_3_Tot.kWh_Tmr,?,?) ,[XIC(VFD_3_Tot.kWh_Tmr.DN) ,XIC(AITot_VFD3.Reset) ,XIC(MIDNIGHT) ] AI_Totalizer(AITot_VFD3,VFD_3_Tot.Power,MIDNIGHT,1,3,1,2,999999999) ,CPT(VFD_3_Tot.Energy,AITot_VFD3.NonResetTotal/(10**AITot_VFD3.IDP)) ];
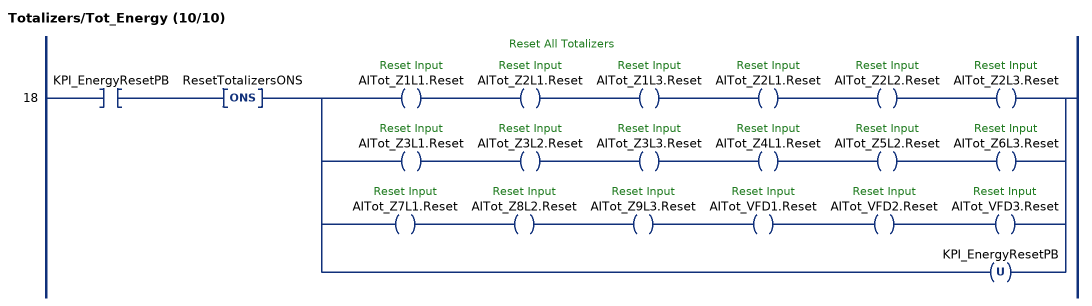
   // Reset All Totalizers
   18: XIC(KPI_EnergyResetPB)ONS(ResetTotalizersONS)[OTE(AITot_Z1L1.Reset) OTE(AITot_Z2L1.Reset) OTE(AITot_Z1L3.Reset) OTE(AITot_Z2L1.Reset) OTE(AITot_Z2L2.Reset) OTE(AITot_Z2L3.Reset) ,OTE(AITot_Z3L1.Reset) OTE(AITot_Z3L2.Reset) OTE(AITot_Z3L3.Reset) OTE(AITot_Z4L1.Reset) OTE(AITot_Z5L2.Reset) OTE(AITot_Z6L3.Reset) ,OTE(AITot_Z7L1.Reset) OTE(AITot_Z8L2.Reset) OTE(AITot_Z9L3.Reset) OTE(AITot_VFD1.Reset) OTE(AITot_VFD2.Reset) OTE(AITot_VFD3.Reset) ,OTU(KPI_EnergyResetPB) ];
END_ROUTINE
END_PROGRAM
